FUNCTION functie : BOOL
VAR_INPUT
	Spoelen_start : BOOL;
	Timer : TON;
END_VAR
VAR
	

END_VAR


// machine word gespoeld wanneer die in stap 10 is van proces_1

GVL.Spoelen_machine := TRUE;

		IF Timer.Q = TRUE THEN
			Timer(IN:=FALSE);
			functie := TRUE;
			GVL.Spoelen_machine := FALSE;
		END_IF

END_FUNCTION

(* stored: Version 1.1.0.1, ProductVersion 3.1.4024.12
   POU functie: Id {aeb3075e-9858-42cb-9531-a1dc2ef35f12}, SpecialFunc None *)
